(* IEC 61131-3 sources: Berechnungsplattform/PLC_CODESYS/CAN_Communication, 1 file *)

(* ---- CAN_Interface.st ---- *)
(* ============================================================================
   CAN Interface for Intercontrol DIGSY Fusion S
   Development Environment: CODESYS
   Description: CAN bus communication function block for receiving and
                transmitting CAN messages
   ============================================================================ *)

TYPE CAN_Message :
STRUCT
    ID          : DWORD;        (* CAN Identifier (11-bit or 29-bit) *)
    DLC         : BYTE;         (* Data Length Code (0-8) *)
    Data        : ARRAY[0..7] OF BYTE;  (* CAN Data bytes *)
    Extended    : BOOL;         (* TRUE = 29-bit ID, FALSE = 11-bit ID *)
    RTR         : BOOL;         (* Remote Transmission Request *)
    Timestamp   : TIME;         (* Timestamp of message *)
END_STRUCT
END_TYPE

TYPE CAN_Status :
(
    CAN_STATUS_OK := 0,
    CAN_STATUS_ERROR := 1,
    CAN_STATUS_BUSY := 2,
    CAN_STATUS_TIMEOUT := 3,
    CAN_STATUS_BUFFER_FULL := 4,
    CAN_STATUS_NOT_INITIALIZED := 5
);
END_TYPE

(* ============================================================================
   FUNCTION_BLOCK: FB_CAN_Interface
   Description: Main CAN interface function block for DIGSY Fusion S
   ============================================================================ *)
FUNCTION_BLOCK FB_CAN_Interface
VAR_INPUT
    bEnable             : BOOL := FALSE;    (* Enable CAN interface *)
    dwBaudrate          : DWORD := 250000;  (* CAN Baudrate in bit/s *)
    bSendMessage        : BOOL := FALSE;    (* Trigger to send message *)
    stTxMessage         : CAN_Message;      (* Message to transmit *)
END_VAR

VAR_OUTPUT
    bInitialized        : BOOL := FALSE;    (* CAN interface initialized *)
    bMessageReceived    : BOOL := FALSE;    (* New message received *)
    stRxMessage         : CAN_Message;      (* Last received message *)
    eStatus             : CAN_Status;       (* Current CAN status *)
    dwTxCounter         : DWORD := 0;       (* Transmitted message counter *)
    dwRxCounter         : DWORD := 0;       (* Received message counter *)
    dwErrorCounter      : DWORD := 0;       (* Error counter *)
END_VAR

VAR
    bInitDone           : BOOL := FALSE;
    bSendTrigger        : BOOL := FALSE;
    bPrevSendMessage    : BOOL := FALSE;
    tTimeout            : TON;
    tWatchdog           : TON;
    dwInternalState     : DWORD := 0;
END_VAR

(* Main execution *)
IF NOT bEnable THEN
    bInitialized := FALSE;
    bInitDone := FALSE;
    eStatus := CAN_STATUS_NOT_INITIALIZED;
    dwInternalState := 0;
    RETURN;
END_IF

(* State machine for CAN initialization and operation *)
CASE dwInternalState OF
    0: (* Initialization state *)
        (* Initialize CAN controller with baudrate *)
        (* NOTE: Hardware-specific initialization for DIGSY Fusion S
           Replace the following placeholder with actual DIGSY Fusion S CAN library calls:

           Example using Intercontrol CAN library:
           - CAN_Init(channel := 0, baudrate := dwBaudrate);
           - Configure CAN filters as needed

           The actual implementation depends on the specific DIGSY Fusion S
           firmware version and installed CAN libraries. Consult the
           Intercontrol documentation for the correct function calls.
        *)

        (* Placeholder: Set initialized flag after hardware init *)
        bInitDone := TRUE;
        bInitialized := TRUE;
        eStatus := CAN_STATUS_OK;
        dwInternalState := 1;

    1: (* Normal operation state *)
        (* Check for incoming messages *)
        (* NOTE: Hardware-specific CAN receive for DIGSY Fusion S
           Replace with actual CAN library calls, for example:

           IF CAN_Receive(channel := 0, msg => stRxMessage) THEN
               bMessageReceived := TRUE;
               dwRxCounter := dwRxCounter + 1;
           ELSE
               bMessageReceived := FALSE;
           END_IF

           The exact function names depend on the DIGSY Fusion S CAN library.
           Common libraries include:
           - Intercontrol CAN Driver Library
           - CANopen Stack (if using CANopen protocol)
           - Raw CAN access functions
        *)

        (* Detect rising edge on send trigger *)
        bSendTrigger := bSendMessage AND NOT bPrevSendMessage;
        bPrevSendMessage := bSendMessage;

        IF bSendTrigger THEN
            (* Transmit message *)
            (* NOTE: Hardware-specific CAN transmit for DIGSY Fusion S
               Replace with actual CAN library calls, for example:

               IF CAN_Transmit(channel := 0, msg := stTxMessage) THEN
                   dwTxCounter := dwTxCounter + 1;
               ELSE
                   dwErrorCounter := dwErrorCounter + 1;
                   eStatus := CAN_STATUS_ERROR;
               END_IF

               Ensure proper error handling for transmission failures.
            *)
            dwTxCounter := dwTxCounter + 1;
        END_IF

        (* Timeout watchdog *)
        tWatchdog(IN := TRUE, PT := T#1S);
        IF tWatchdog.Q THEN
            tWatchdog(IN := FALSE);
            (* Watchdog reset - communication alive check *)
        END_IF

    ELSE
        (* Error state - reset to initialization *)
        dwInternalState := 0;
        dwErrorCounter := dwErrorCounter + 1;
        eStatus := CAN_STATUS_ERROR;
END_CASE

END_FUNCTION_BLOCK

(* ============================================================================
   FUNCTION_BLOCK: FB_CAN_MessageFilter
   Description: CAN message filter for specific CAN IDs
   ============================================================================ *)
FUNCTION_BLOCK FB_CAN_MessageFilter
VAR_INPUT
    stInMessage         : CAN_Message;      (* Input CAN message *)
    bNewMessage         : BOOL := FALSE;    (* New message trigger *)
    dwFilterID          : DWORD := 0;       (* Filter CAN ID *)
    dwFilterMask        : DWORD := 16#7FF;  (* Filter mask (default: all bits) *)
END_VAR

VAR_OUTPUT
    bMatch              : BOOL := FALSE;    (* Message matches filter *)
    stOutMessage        : CAN_Message;      (* Filtered output message *)
END_VAR

(* Check if incoming message matches filter *)
IF bNewMessage THEN
    IF (stInMessage.ID AND dwFilterMask) = (dwFilterID AND dwFilterMask) THEN
        bMatch := TRUE;
        stOutMessage := stInMessage;
    ELSE
        bMatch := FALSE;
    END_IF
ELSE
    bMatch := FALSE;
END_IF

END_FUNCTION_BLOCK
